VAR_GLOBAL
	FirstCycle				:BOOL:=TRUE;
	Clock_1_Hz				:FB_Clock;
	LiveBit					:FB_LiveBit;
END_VAR

(* stored: Version 1.1.0.1, ProductVersion 3.1.0.36
   GVL GVL_Main: Id {d8992863-d5dc-4a74-9d03-791e5077aabe} *)
